# EPICS substitutions: apps/CaenHVApp/Db/CaenHV_crate12.substitutions
file "db/AS503_Chan.template" {
pattern
    {P,      H,  S,   V}
    {hchv,  12,  00,  000}
    {hchv,  12,  00,  001}
    {hchv,  12,  00,  002}
    {hchv,  12,  00,  003}
    {hchv,  12,  00,  004}
    {hchv,  12,  00,  005}
    {hchv,  12,  00,  006}
    {hchv,  12,  00,  007}
    {hchv,  12,  00,  008}
    {hchv,  12,  00,  009}
    {hchv,  12,  00,  010}
    {hchv,  12,  00,  011}
    {hchv,  12,  00,  012}
    {hchv,  12,  00,  013}
    {hchv,  12,  00,  014}
    {hchv,  12,  00,  015}
}
file "db/AS503_Chan.template" {
pattern
    {P,      H,  S,   V}
    {hchv,  12,  01, 000}
    {hchv,  12,  01, 001}
    {hchv,  12,  01, 002}
    {hchv,  12,  01, 003}
    {hchv,  12,  01, 004}
    {hchv,  12,  01, 005}
    {hchv,  12,  01, 006}
    {hchv,  12,  01, 007}
    {hchv,  12,  01, 008}
    {hchv,  12,  01, 009}
    {hchv,  12,  01, 010}
    {hchv,  12,  01, 011}
    {hchv,  12,  01, 012}
    {hchv,  12,  01, 013}
    {hchv,  12,  01, 014}
    {hchv,  12,  01, 015}
}
file "db/AS503_Chan.template" {
pattern
    {P,      H,  S,   V}
    {hchv,  12,  02, 000}
    {hchv,  12,  02, 001}
    {hchv,  12,  02, 002}
    {hchv,  12,  02, 003}
    {hchv,  12,  02, 004}
    {hchv,  12,  02, 005}
    {hchv,  12,  02, 006}
    {hchv,  12,  02, 007}
    {hchv,  12,  02, 008}
    {hchv,  12,  02, 009}
    {hchv,  12,  02, 010}
    {hchv,  12,  02, 011}
    {hchv,  12,  02, 012}
    {hchv,  12,  02, 013}
    {hchv,  12,  02, 014}
    {hchv,  12,  02, 015}
}
file "db/AS503_Chan.template" {
pattern
    {P,      H,  S,   V}
    {hchv,  12,  03, 000}
    {hchv,  12,  03, 001}
    {hchv,  12,  03, 002}
    {hchv,  12,  03, 003}
    {hchv,  12,  03, 004}
    {hchv,  12,  03, 005}
    {hchv,  12,  03, 006}
    {hchv,  12,  03, 007}
    {hchv,  12,  03, 008}
    {hchv,  12,  03, 009}
    {hchv,  12,  03, 010}
    {hchv,  12,  03, 011}
    {hchv,  12,  03, 012}
    {hchv,  12,  03, 013}
    {hchv,  12,  03, 014}
    {hchv,  12,  03, 015}
}
